{attribute 'GeneratedUsingTerminal: EJ6224-0000-0016'}
{attribute addProperty BoxType "EJ6224-0000-0016"}
{attribute addProperty Id "Module_1_DeviceState_Inputs_DeviceModule_1_DeviceState_Inputs_Device_5322301C2Module_2_DeviceState_InputsModule_2_DeviceState_Inputs_BD6C70354WcStateAT %I*WcState_9091E0EB2InfoDataAT %I*InfoData_41C547A32"}
{attribute addProperty CRC "564608256"}
{attribute addProperty Size "10"}
TYPE EJ6224_21A73D00 EXTENDS EtcSlaveTerminalBase_947E5A46 :
STRUCT
	{attribute addProperty Name "Module_1_DeviceState_Inputs_Device"}
	Module_1_DeviceState_Inputs_Device : Module_1_DeviceState_Inputs_Device_5322301C;
	{attribute addProperty Name "Module_2_DeviceState_Inputs"}
	Module_2_DeviceState_Inputs : Module_2_DeviceState_Inputs_BD6C7035;
	{attribute addProperty Name "WcState"}
	WcState : WcState_9091E0EB;
	{attribute addProperty Name "InfoData"}
	InfoData : InfoData_41C547A3;
END_STRUCT
END_TYPE

(* stored: Version 1.2.0.0, ProductVersion 3.1.4024.9
   DUT EJ6224_21A73D00: Id {0bc1228c-22de-48f9-a562-9559ef1590a1} *)
